(* LS Electric XG5000 project: Stride_IOLink_EIP_FB *)
(* project contains a function block for communicating with Automationdirect's IO-Link masters *)
(* PLC LSPLC *)
(* module base 0 slot 0: Input/Output Module:XEM-DN/DP32HP (DC 24V Input, Transistor Output, 32 Contacts) *)
(* module base 0 slot 1: Internal Positioning:XBF-PO06E (Open Collector Type, 6 Axis) *)
(* module base 0 slot 2: EtherNet/IP:XBL-EIPT (EtherNet/IP communication module, electrical) *)
VAR_GLOBAL
    Stride_IOLink_Input00 : ARRAY[0..393] OF BYTE; (* Input data for IO-Link master *)
    Stride_IOLink_Output00 : ARRAY[0..259] OF BYTE; (* Output data for IO-Link master *)
END_VAR

TYPE Contrinex_RLH_RFID_UDT : (* data type for Contrinex RLH-xxxPA-NIS RFID reader/writer with IO-Link interface. *)
STRUCT
    Status_Ready : BOOL; (* Will toggle state when command executed and new data is available *)
    Status_Error : BOOL; (* Command executed with error. *)
    Status_Tag_Present : BOOL; (* Tag present in range of transponder *)
    Status_Antenna_On : BOOL; (* Transponder antenna is powered *)
    Status_RSSI_Level : USINT; (* Signal level between transponder and tag. *)
    Status_Error_Code : USINT; (* ISO 15693 error code. 1: CommandNotSupported. 2: FormatError. 3: OptionNotSupported. 5: CommandProblem. 6: CommTagError. 15:TagError. 16: NoMemoryBlock. 18: BlockProtected. 27:AppLOGError. 30: TAGCommError. 255: AppGeneralError. *)
    Status_Alarm_1 : BOOL; (* Alarm1 active *)
    Status_Alarm_2 : BOOL; (* Alarm 2 active *)
    Status_Address : USINT; (* First transponder memory block address where the R/W command was executed *)
    Status_Command_Feedback : USINT; (* Feedback of command sent to transponder *)
    Status_Tag_UID : ARRAY[0..7] OF BYTE; (* Transponder unique ID number *)
    Status_Tag_In_Range_Time : DINT; (* Transponder in-range time in milliseconds *)
    Status_Tag_In_Range_Start_Time : DINT; (* Transponder in-range system start time in milliseconds *)
    Status_Ready_Last_Scan : BOOL; (* Last Scan Data for determining change of ready bit. *)
    Status_Read_Tag_Value : ARRAY[0..30] OF BYTE; (* data read from userspace on tag *)
    Control_Set_Tag_Value : ARRAY[0..30] OF BYTE; (* data to write to userspace on tag *)
    Received_Tag_ASCII : STRING; (* received transponder data, converted to ASCII for readability *)
    Set_Tag_ASCII : STRING; (* Optional ASCII string to send to transponder if readable text is desired. *)
    Control_Start_Operation : BOOL; (* Toggle to begin desired RFID operation (not used for Auto-Read or Auto-Write) *)
    Control_Switch_Off_Antenna : BOOL; (* Disables antenna when high *)
    Control_Command : USINT; (* command to send to transponder *)
    Control_NB_Block : USINT; (* number of transponder memory block to R/W *)
    Control_Address : USINT; (* first transponder memory block address where the R/W command will be executed. *)
    Control_Mode_Set_None : BOOL; (* Set to High to disable RFID functions *)
    Control_Mode_Set_Auto_Read : BOOL; (* Set to high to enable auto-read function. *)
    Control_Mode_Set_Auto_Write : BOOL; (* Set to high to enable auto-write function *)
    Control_Mode_Set_Read : BOOL; (* Set to high to attempt one single read *)
    Control_Mode_Set_Write : BOOL; (* Set to high to attempt one single write *)
    Control_Mode_Set_Read_Sys : BOOL; (* Set to high to enable tag UID and timings function *)
    Scans_Since_Tag_Last_Seen : UINT; (* Counter value to watch for absence of tag. *)
END_STRUCT;
END_TYPE

TYPE Murr_DIO_Hub_UDT : (* user data type for the Murrelektronik MVP12/MVP8 Digital Input/Output IO-Link hub *)
STRUCT
    Digital_Input : ARRAY[0..15] OF BOOL; (* Mapped Digital Inputs *)
    Digital_Output : ARRAY[0..15] OF BOOL; (* Mapped Digital Outputs *)
    Fault_Present : BOOL; (* Active if there is a fault with MURR dio hub *)
    Fault_IO_Point : INT; (* ID of channel experiencing a fault *)
END_STRUCT;
END_TYPE

TYPE Stride_IOLink_Port_UDT :
STRUCT
    Vendor_ID : UINT; (* IO-Link Vendor ID *)
    Device_ID : DINT; (* IO-Link Device ID *)
    Port_Status_Operate : BOOL; (* 1 = device is connected and active *)
    Port_Status_Error : BOOL; (* 1 = error or warning has occurred on this port *)
    Port_Status_Valid : BOOL; (* 1 = process data is valid *)
    Discrete_Input : ARRAY[0..1] OF BOOL; (* Physical Input pins *)
    Discrete_Output : ARRAY[0..1] OF BOOL; (* Physical Output pins *)
    Cyclic_Data_In : ARRAY[0..31] OF BYTE; (* process data from IO-Link device. *)
    Cyclic_Data_Out : ARRAY[0..31] OF BYTE; (* Control data to IO-Link device. *)
END_STRUCT;
END_TYPE

FUNCTION_BLOCK Contrinex_RFID_FB
(* Function block for Contrinex RLH-xxxPA-NIS RFID system *)
VAR_INPUT
    Enable : BOOL; (* Enable for function block *)
    Copy_SetTagASCII_to_ControlSetValue : BOOL; (* this will enable copying UserRFID.Set_Tag_ASCII to UserRFID.Control.Set_Tag_Value. *)
END_VAR
VAR_IN_OUT
    User_RFID : Contrinex_RLH_RFID_UDT; (* Data type for the Contrinex RFID module *)
    Port : Stride_IOLink_Port_UDT; (* variable for IO-Link master port. *)
END_VAR
VAR_OUTPUT
    Active : BOOL; (* Function block is active. *)
END_VAR
VAR
    InTemp : ARRAY[0..31] OF BYTE; (* temporary input array *)
    OutTemp : ARRAY[0..31] OF BYTE; (* temporary output array *)
    tempBool : BOOL; (* temporary bool storage *)
    tempDWord1 : DWORD; (* temporary dword storage *)
    tempWord1 : WORD; (* temporary word storage *)
    tempWord2 : WORD; (* temporary word storage *)
END_VAR
(*
AutomationDirect.com has provided this code for convenience. This sample code is provided "as-is" with no expressed or implied warranty and has not been thoroughly tested for all conditions and environments.  
While AutomationDirect.com makes every effort to provide error-free code that can be used as-is, it is the user's responsibility to completely test this code in operation to ensure it meets all system and safety requirements for the intended application or system.
 By loading and running this code, you are acknowledging the responsibility to completely test the code in your system before deployment.
*)
(***************************************************************************************************
	The 'Contrinex_RFID_FB' function block use one of the Port_X0 thru Port_X7 from Stride_IOLink_Master_FB.
		This function block separates the source data buffers for a Contrinex RLH RFID module that is connected to the given Port_XX that is passed in.
						
	***************************************************************************************************)
	
	IF (Enable = TRUE) THEN
		Active := TRUE;
		
		(* Map Status variables *)
		InTemp := ARY_MOVE(MOVE_NUM:=31, IN:=Port.Cyclic_Data_In, IN_INDX:=0, OUT_INDX:=0);
		
		User_RFID.Status_Command_Feedback.0  := InTemp[0].0;
		User_RFID.Status_Command_Feedback.1  := InTemp[0].1;
		User_RFID.Status_Command_Feedback.2  := InTemp[0].2;
		User_RFID.Status_Antenna_On  := InTemp[0].4;
		User_RFID.Status_Tag_Present  := InTemp[0].5;
		User_RFID.Status_Error  := InTemp[0].6;
		User_RFID.Status_Ready  := InTemp[0].7;
		
		User_RFID.Status_Alarm_1  := InTemp[1].0;
		User_RFID.Status_Alarm_2  := InTemp[1].1;
		User_RFID.Status_Error_Code.0  := InTemp[1].2;
		User_RFID.Status_Error_Code.1  := InTemp[1].3;
		User_RFID.Status_Error_Code.2  := InTemp[1].4;
		User_RFID.Status_Error_Code.3  := InTemp[1].5;
		User_RFID.Status_Error_Code.4  := InTemp[1].6;
		User_RFID.Status_Error_Code.5  := InTemp[1].7;
		
		User_RFID.Status_RSSI_Level :=  BYTE_TO_USINT(InTemp[2]);
		User_RFID.Status_Address := BYTE_TO_USINT(InTemp[3]);
		
		
		//control mode commands.
		IF (User_RFID.Control_Mode_Set_None = TRUE) THEN
			User_RFID.Control_Command := 0;
			User_RFID.Control_Mode_Set_None := FALSE;
		
		ELSIF (User_RFID.Control_Mode_Set_Auto_Read = TRUE) THEN
			User_RFID.Control_Command := 1;
			User_RFID.Control_Mode_Set_Auto_Read := FALSE;
		
		ELSIF (User_RFID.Control_Mode_Set_Auto_Write = TRUE) THEN
			User_RFID.Control_Command := 2;	
			User_RFID.Control_Mode_Set_Auto_Write := FALSE;
			
		ELSIF (User_RFID.Control_Mode_Set_Read = TRUE) THEN
			User_RFID.Control_Command := 3;		
			User_RFID.Control_Mode_Set_Read := FALSE;
		
		ELSIF ( User_RFID.Control_Mode_Set_Write = TRUE) THEN
			User_RFID.Control_Command := 4;		
		  	User_RFID.Control_Mode_Set_Write :=  FALSE;
		  	
		  ELSIF(User_RFID.Control_Mode_Set_Read_Sys = TRUE) THEN
		  	User_RFID.Control_Command := 5;	
		    User_RFID.Control_Mode_Set_Read_Sys := FALSE;
		    
		   END_IF; 
		
		//update last read tag when new data available.
		IF (User_RFID.Status_Command_Feedback = 1 OR User_RFID.Status_Command_Feedback = 3) AND ( (User_RFID.Status_Ready = TRUE AND User_RFID.Status_Ready_Last_Scan = FALSE) OR (User_RFID.Status_Ready_Last_Scan = TRUE AND User_RFID.Status_Ready = FALSE) ) THEN
			User_RFID.Status_Read_Tag_Value := ARY_MOVE(MOVE_NUM:=28, IN:=InTemp, IN_INDX:=4, OUT_INDX:=0);
		END_IF;
		
		//Convert received tag data to ASCII
		User_RFID.Received_Tag_ASCII :=BYTE_STRING(IN:=User_RFID.Status_Read_Tag_Value);
		
		
		//calculate 'tag-in-range' times and read tag UID
		IF (User_RFID.Status_Command_Feedback = 5) THEN
			
			tempWord1 := BYTE_WORD(LOW:=InTemp[27], HIGH:=InTemp[26]);
			tempWord2 :=BYTE_WORD(LOW:=InTemp[25], HIGH:=InTemp[24]);
			tempDWord1 := WORD_DWORD(LOW:=tempWord1, HIGH:= tempWord2);
			User_RFID.Status_Tag_In_Range_Time := DWORD_TO_DINT(IN:= tempDWord1);
			
			tempWord1 := BYTE_WORD(LOW:=InTemp[19], HIGH:=InTemp[18]);
			tempWord2 :=BYTE_WORD(LOW:=InTemp[17], HIGH:=InTemp[16]);
			tempDWord1 := WORD_DWORD(LOW:=tempWord1, HIGH:= tempWord2);
			User_RFID.Status_Tag_In_Range_Start_Time := DWORD_TO_DINT(IN:= tempDWord1);
			
			User_RFID.Status_Tag_UID := ARY_MOVE(MOVE_NUM:=8, IN:=InTemp, IN_INDX:=5, OUT_INDX:=0);
			
		END_IF;
		
		
		//Clear read tag data when tag isn't present for 50 scans
		IF (User_RFID.Status_Tag_Present = TRUE) THEN
			User_RFID.Scans_Since_Tag_Last_Seen := 0;
		ELSE
			User_RFID.Scans_Since_Tag_Last_Seen := User_RFID.Scans_Since_Tag_Last_Seen + 1;
		END_IF;
		
		IF (User_RFID.Scans_Since_Tag_Last_Seen > 50) THEN
			tempBool := ARY_FLL(DATA:=0, SRC:=User_RFID.Status_Read_Tag_Value, INDX:=0, LEN:=28);
			tempBool := ARY_FLL(DATA:=0, SRC:=User_RFID.Status_Tag_UID, INDX:=0, LEN:=8);
		END_IF;
		
		
		//when write command active, copy desired tag value to output data
		IF (User_RFID.Status_Command_Feedback =  4) OR (User_RFID.Status_Command_Feedback = 2) THEN
			OutTemp := ARY_MOVE(MOVE_NUM:=28, IN:=User_RFID.Control_Set_Tag_Value, IN_INDX:=0, OUT_INDX:=4); 
		END_IF;
		
		//copy string into set array if enabled
		IF (Copy_SetTagASCII_to_ControlSetValue = TRUE) THEN
			User_RFID.Control_Set_Tag_Value :=STRING_BYTE(IN:=User_RFID.Set_Tag_ASCII);
		END_IF;	
		
		//Pack commands into first command byte.
		OutTemp[0].0  := User_RFID.Control_Command.0;
		OutTemp[0].1  := User_RFID.Control_Command.1;
		OutTemp[0].2  := User_RFID.Control_Command.2;
		OutTemp[0].4  := User_RFID.Control_Switch_Off_Antenna;
		OutTemp[0].7  := User_RFID.Control_Start_Operation;
		
		
		//pack memory block target size into second command byte.
		OutTemp[1].0  := User_RFID.Control_NB_Block.0;
		OutTemp[1].1  := User_RFID.Control_NB_Block.1;
		OutTemp[1].2  := User_RFID.Control_NB_Block.2;
		
		//copy target memory address start point into fourth command byte
		OutTemp[3]  := USINT_TO_BYTE(User_RFID.Control_Address);
		
		//copy tag ready bit value to last-scan value
		User_RFID.Status_Ready_Last_Scan :=  User_RFID.Status_Ready;
		
		//map outputs to port
		Port.Cyclic_Data_Out := ARY_MOVE(MOVE_NUM:=32, IN:=OutTemp, IN_INDX:=0, OUT_INDX:=0);
	
		
	ELSE
		Active := FALSE;
		
	END_IF;
END_FUNCTION_BLOCK

FUNCTION_BLOCK Murr_DIO_Hub_FB
(* function block for mapping data from Murrelektronik MVP12/MVP8 Digital Input/Output IO-Link hub *)
VAR_INPUT
    Enable : BOOL; (* enable function block *)
END_VAR
VAR_IN_OUT
    DIO_Hub : Murr_DIO_Hub_UDT; (* variable for MURR DIO Hub *)
    Port : Stride_IOLink_Port_UDT; (* variable for IO-Link master port. *)
END_VAR
VAR_OUTPUT
    Active : BOOL; (* function block is active *)
END_VAR
VAR
    InTemp : ARRAY[0..31] OF BYTE; (* temporary input array *)
    OutTemp : ARRAY[0..31] OF BYTE; (* temporary output array *)
END_VAR
(*
AutomationDirect.com has provided this code for convenience. This sample code is provided "as-is" with no expressed or implied warranty and has not been thoroughly tested for all conditions and environments.  
While AutomationDirect.com makes every effort to provide error-free code that can be used as-is, it is the user's responsibility to completely test this code in operation to ensure it meets all system and safety requirements for the intended application or system.
 By loading and running this code, you are acknowledging the responsibility to completely test the code in your system before deployment.
*)
(***************************************************************************************************
	The 'Murr_DIO_Hub_FB' function block use one of the Port_X0 thru Port_X7 from Stride_IOLink_Master_FB.
		This function block separates the source data buffers for a Murr DIO Hub that is connected to the given Port_XX that is passed in.
						
	***************************************************************************************************)
	
IF (Enable = TRUE) THEN		
	Active := TRUE;
	
	//map inputs
	InTemp := ARY_MOVE(MOVE_NUM:=31, IN:=Port.Cyclic_Data_In, IN_INDX:=0, OUT_INDX:=0);
	
	DIO_Hub.Digital_Input[0] := InTemp[0].0;
	DIO_Hub.Digital_Input[1] := InTemp[0].1;
	DIO_Hub.Digital_Input[2] := InTemp[0].2;
	DIO_Hub.Digital_Input[3] := InTemp[0].3;
	DIO_Hub.Digital_Input[4] := InTemp[0].4;
	DIO_Hub.Digital_Input[5] := InTemp[0].5;
	DIO_Hub.Digital_Input[6] := InTemp[0].6;
	DIO_Hub.Digital_Input[7] := InTemp[0].7;
	DIO_Hub.Digital_Input[8] := InTemp[1].0;
	DIO_Hub.Digital_Input[9] := InTemp[1].1;
	DIO_Hub.Digital_Input[10] := InTemp[1].2;
	DIO_Hub.Digital_Input[11] := InTemp[1].3;
	DIO_Hub.Digital_Input[12] := InTemp[1].4;
	DIO_Hub.Digital_Input[13] := InTemp[1].5;
	DIO_Hub.Digital_Input[14] := InTemp[1].6;
	DIO_Hub.Digital_Input[15] := InTemp[1].7;	
	
	DIO_Hub.Fault_Present := InTemp[2].0;
	
	// map io point number that has a fault
	DIO_Hub.Fault_IO_Point.0 := InTemp[2].3;
	DIO_Hub.Fault_IO_Point.1 := InTemp[2].4;
	DIO_Hub.Fault_IO_Point.2 := InTemp[2].5;
	DIO_Hub.Fault_IO_Point.3 := InTemp[2].6;
	
	//map outputs from DIO Hub to OutTemp
	OutTemp[0].0 := DIO_Hub.Digital_Output[0];
	OutTemp[0].1 := DIO_Hub.Digital_Output[1];
	OutTemp[0].2 := DIO_Hub.Digital_Output[2];
	OutTemp[0].3 := DIO_Hub.Digital_Output[3];
	OutTemp[0].4 := DIO_Hub.Digital_Output[4];
	OutTemp[0].5 := DIO_Hub.Digital_Output[5];
	OutTemp[0].6 := DIO_Hub.Digital_Output[6];
	OutTemp[0].7 := DIO_Hub.Digital_Output[7];
	OutTemp[1].0 := DIO_Hub.Digital_Output[8];
	OutTemp[1].1 := DIO_Hub.Digital_Output[9];
	OutTemp[1].2 := DIO_Hub.Digital_Output[10];
	OutTemp[1].3 := DIO_Hub.Digital_Output[11];
	OutTemp[1].4 := DIO_Hub.Digital_Output[12];
	OutTemp[1].5 := DIO_Hub.Digital_Output[13];
	OutTemp[1].6 := DIO_Hub.Digital_Output[14];
	OutTemp[1].7 := DIO_Hub.Digital_Output[15];
	
	
	
	
	//map outputs to port
	Port.Cyclic_Data_Out := ARY_MOVE(MOVE_NUM:=32, IN:=OutTemp, IN_INDX:=0, OUT_INDX:=0);
	
	
ELSE
	Active := FALSE;
	
END_IF;
END_FUNCTION_BLOCK

FUNCTION_BLOCK Stride_IOLink_Master_FB
(* function block for mapping data from Stride Ethernet/IP IO-Link master *)
VAR_INPUT
    Enable : BOOL; (* Enable the function block *)
    Source_InputData : ARRAY[0..393] OF BYTE; (* Input data from the EtherNet/IP IO-Link master *)
END_VAR
VAR_IN_OUT
    Source_OutputData : ARRAY[0..259] OF BYTE; (* Output data from the EtherNet/IP IO-Link master *)
    Port_X0 : Stride_IOLink_Port_UDT; (* Port X0 of IO-Link master *)
    Port_X1 : Stride_IOLink_Port_UDT; (* Port X1 of IO-Link master *)
    Port_X2 : Stride_IOLink_Port_UDT; (* Port X2 of IO-Link master *)
    Port_X3 : Stride_IOLink_Port_UDT; (* Port X3 of IO-Link master *)
    Port_X4 : Stride_IOLink_Port_UDT; (* Port X4 of IO-Link master *)
    Port_X5 : Stride_IOLink_Port_UDT; (* Port X5 of IO-Link master *)
    Port_X6 : Stride_IOLink_Port_UDT; (* Port X6 of IO-Link master *)
    Port_X7 : Stride_IOLink_Port_UDT; (* Port X7 of IO-Link master *)
END_VAR
VAR_OUTPUT
    Active : BOOL; (* status that function block is active *)
END_VAR
VAR
    InputStatus : ARRAY[0..7] OF BYTE; (* input status data *)
    InTemp : ARRAY[0..393] OF BYTE; (* temporary input buffer to copy Source_InputData too. *)
    OutTemp : ARRAY[0..259] OF BYTE; (* temporary output buffer to copy to Source_OutputData *)
    WTemp1 : WORD; (* temporary word 1 *)
    WTemp2 : WORD; (* temporary word 2 *)
END_VAR
(*
AutomationDirect.com has provided this code for convenience. This sample code is provided "as-is" with no expressed or implied warranty and has not been thoroughly tested for all conditions and environments.  
While AutomationDirect.com makes every effort to provide error-free code that can be used as-is, it is the user's responsibility to completely test this code in operation to ensure it meets all system and safety requirements for the intended application or system.
 By loading and running this code, you are acknowledging the responsibility to completely test the code in your system before deployment.
*)
(***************************************************************************************************
	The 'Stride_IOLink_Master_FB' function block uses data type BYTE for Source_InputData and Source_OutputData.
		This function block separates the source data buffers into the individual ports of X0 thru X7.
		
									Data type:: BYTE
									Input Size: 394 bytes
									Output Size: 260 bytes
									EDS File: SIOL_EI8B_EIP_Rev_1_1.eds
									
	***************************************************************************************************)
	
IF (Enable = TRUE) THEN		
	Active := TRUE;	
	
	//copy Source_InputData to temporary local one
	InTemp := ARY_MOVE(MOVE_NUM:=394, IN:=Source_InputData, IN_INDX:=0, OUT_INDX:=0);
	

	//Port X0 mapping
	Port_X0.Discrete_Input[0] := InTemp[0].0;
	Port_X0.Discrete_Input[1] := InTemp[0].1;
	OutTemp[0].0 := Port_X0.Discrete_Output[0];
	OutTemp[0].1 :=Port_X0.Discrete_Output[1];
	
	Port_X0.Cyclic_Data_In := ARY_MOVE(MOVE_NUM:=32, IN:=InTemp, IN_INDX:=10, OUT_INDX:=0);
	InputStatus := ARY_MOVE(MOVE_NUM:=8, IN:=InTemp, IN_INDX:=42, OUT_INDX:=0);
	OutTemp := ARY_MOVE(MOVE_NUM:=32, IN:=Port_X0.Cyclic_Data_Out, IN_INDX:=0, OUT_INDX:=2);
	
	Port_X0.Port_Status_Operate := InputStatus[0].5;
	Port_X0.Port_Status_Error :=  InputStatus[0].6;
	Port_X0.Port_Status_Valid := InputStatus[0].7;
	
	Port_X0.Vendor_ID := WORD_TO_UINT(BYTE_WORD(LOW:=InputStatus[2], HIGH:=InputStatus[3]));
	
	WTemp1 := BYTE_WORD(LOW:=InputStatus[4], HIGH:=InputStatus[5]);
	WTemp2 := BYTE_WORD(LOW:=InputStatus[6], HIGH:=InputStatus[7]);
	Port_X0.Device_ID := DWORD_TO_DINT(WORD_DWORD(LOW:=WTemp1, HIGH:=WTemp2));
	
	
	
	//Port X1 mapping
	Port_X1.Discrete_Input[0] := InTemp[0].2;
	Port_X1.Discrete_Input[1] := InTemp[0].3;
	OutTemp[0].2 := Port_X1.Discrete_Output[0];
	OutTemp[0].3 :=Port_X1.Discrete_Output[1];
	
	Port_X1.Cyclic_Data_In := ARY_MOVE(MOVE_NUM:=32, IN:=InTemp, IN_INDX:=50, OUT_INDX:=0);
	InputStatus := ARY_MOVE(MOVE_NUM:=8, IN:=InTemp, IN_INDX:=82, OUT_INDX:=0);
	OutTemp := ARY_MOVE(MOVE_NUM:=32, IN:=Port_X1.Cyclic_Data_Out, IN_INDX:=0, OUT_INDX:=34);
	
	Port_X1.Port_Status_Operate := InputStatus[0].5;
	Port_X1.Port_Status_Error :=  InputStatus[0].6;
	Port_X1.Port_Status_Valid := InputStatus[0].7;
	
	Port_X1.Vendor_ID := WORD_TO_UINT(BYTE_WORD(LOW:=InputStatus[2], HIGH:=InputStatus[3]));
	
	WTemp1 := BYTE_WORD(LOW:=InputStatus[4], HIGH:=InputStatus[5]);
	WTemp2 := BYTE_WORD(LOW:=InputStatus[6], HIGH:=InputStatus[7]);
	Port_X1.Device_ID := DWORD_TO_DINT(WORD_DWORD(LOW:=WTemp1, HIGH:=WTemp2));	
	
	
	
	//Port X2 mapping
	Port_X2.Discrete_Input[0] := InTemp[0].4;
	Port_X2.Discrete_Input[1] := InTemp[0].5;
	OutTemp[0].4 := Port_X2.Discrete_Output[0];
	OutTemp[0].5 :=Port_X2.Discrete_Output[1];
	
	Port_X2.Cyclic_Data_In := ARY_MOVE(MOVE_NUM:=32, IN:=InTemp, IN_INDX:=90, OUT_INDX:=0);
	InputStatus := ARY_MOVE(MOVE_NUM:=8, IN:=InTemp, IN_INDX:=122, OUT_INDX:=0);
	OutTemp := ARY_MOVE(MOVE_NUM:=32, IN:=Port_X2.Cyclic_Data_Out, IN_INDX:=0, OUT_INDX:=66);
	
	Port_X2.Port_Status_Operate := InputStatus[0].5;
	Port_X2.Port_Status_Error :=  InputStatus[0].6;
	Port_X2.Port_Status_Valid := InputStatus[0].7;
	
	Port_X2.Vendor_ID := WORD_TO_UINT(BYTE_WORD(LOW:=InputStatus[2], HIGH:=InputStatus[3]));
	
	WTemp1 := BYTE_WORD(LOW:=InputStatus[4], HIGH:=InputStatus[5]);
	WTemp2 := BYTE_WORD(LOW:=InputStatus[6], HIGH:=InputStatus[7]);
	Port_X2.Device_ID := DWORD_TO_DINT(WORD_DWORD(LOW:=WTemp1, HIGH:=WTemp2));	
	
	
	
	//Port X3 mapping
	Port_X3.Discrete_Input[0] := InTemp[0].6;
	Port_X3.Discrete_Input[1] := InTemp[0].7;
	OutTemp[0].6 := Port_X3.Discrete_Output[0];
	OutTemp[0].7 :=Port_X3.Discrete_Output[1];
	
	Port_X3.Cyclic_Data_In := ARY_MOVE(MOVE_NUM:=32, IN:=InTemp, IN_INDX:=130, OUT_INDX:=0);
	InputStatus := ARY_MOVE(MOVE_NUM:=8, IN:=InTemp, IN_INDX:=162, OUT_INDX:=0);
	OutTemp := ARY_MOVE(MOVE_NUM:=32, IN:=Port_X3.Cyclic_Data_Out, IN_INDX:=0, OUT_INDX:=98);
	
	Port_X3.Port_Status_Operate := InputStatus[0].5;
	Port_X3.Port_Status_Error :=  InputStatus[0].6;
	Port_X3.Port_Status_Valid := InputStatus[0].7;
	
	Port_X3.Vendor_ID := WORD_TO_UINT(BYTE_WORD(LOW:=InputStatus[2], HIGH:=InputStatus[3]));
	
	WTemp1 := BYTE_WORD(LOW:=InputStatus[4], HIGH:=InputStatus[5]);
	WTemp2 := BYTE_WORD(LOW:=InputStatus[6], HIGH:=InputStatus[7]);
	Port_X3.Device_ID := DWORD_TO_DINT(WORD_DWORD(LOW:=WTemp1, HIGH:=WTemp2));	
	
	
	
	//Port X4 mapping
	Port_X4.Discrete_Input[0] := InTemp[1].0;
	Port_X4.Discrete_Input[1] := InTemp[1].1;
	OutTemp[1].0 := Port_X4.Discrete_Output[0];
	OutTemp[1].1 :=Port_X4.Discrete_Output[1];
	
	Port_X4.Cyclic_Data_In := ARY_MOVE(MOVE_NUM:=32, IN:=InTemp, IN_INDX:=170, OUT_INDX:=0);
	InputStatus := ARY_MOVE(MOVE_NUM:=8, IN:=InTemp, IN_INDX:=202, OUT_INDX:=0);
	OutTemp := ARY_MOVE(MOVE_NUM:=32, IN:=Port_X4.Cyclic_Data_Out, IN_INDX:=0, OUT_INDX:=130);
	
	Port_X4.Port_Status_Operate := InputStatus[0].5;
	Port_X4.Port_Status_Error :=  InputStatus[0].6;
	Port_X4.Port_Status_Valid := InputStatus[0].7;
	
	Port_X4.Vendor_ID := WORD_TO_UINT(BYTE_WORD(LOW:=InputStatus[2], HIGH:=InputStatus[3]));
	
	WTemp1 := BYTE_WORD(LOW:=InputStatus[4], HIGH:=InputStatus[5]);
	WTemp2 := BYTE_WORD(LOW:=InputStatus[6], HIGH:=InputStatus[7]);
	Port_X4.Device_ID := DWORD_TO_DINT(WORD_DWORD(LOW:=WTemp1, HIGH:=WTemp2));		
	
	
	
	//Port X5 mapping
	Port_X5.Discrete_Input[0] := InTemp[1].2;
	Port_X5.Discrete_Input[1] := InTemp[1].3;
	OutTemp[1].2 := Port_X5.Discrete_Output[0];
	OutTemp[1].3 :=Port_X5.Discrete_Output[1];
	
	Port_X5.Cyclic_Data_In := ARY_MOVE(MOVE_NUM:=32, IN:=InTemp, IN_INDX:=210, OUT_INDX:=0);
	InputStatus := ARY_MOVE(MOVE_NUM:=8, IN:=InTemp, IN_INDX:=242, OUT_INDX:=0);
	OutTemp := ARY_MOVE(MOVE_NUM:=32, IN:=Port_X5.Cyclic_Data_Out, IN_INDX:=0, OUT_INDX:=162);
	
	Port_X5.Port_Status_Operate := InputStatus[0].5;
	Port_X5.Port_Status_Error :=  InputStatus[0].6;
	Port_X5.Port_Status_Valid := InputStatus[0].7;
	
	Port_X5.Vendor_ID := WORD_TO_UINT(BYTE_WORD(LOW:=InputStatus[2], HIGH:=InputStatus[3]));
	
	WTemp1 := BYTE_WORD(LOW:=InputStatus[4], HIGH:=InputStatus[5]);
	WTemp2 := BYTE_WORD(LOW:=InputStatus[6], HIGH:=InputStatus[7]);
	Port_X5.Device_ID := DWORD_TO_DINT(WORD_DWORD(LOW:=WTemp1, HIGH:=WTemp2));	
	

	//Port X6 mapping
	Port_X6.Discrete_Input[0] := InTemp[1].4;
	Port_X6.Discrete_Input[1] := InTemp[1].5;
	OutTemp[1].4 := Port_X6.Discrete_Output[0];
	OutTemp[1].5 :=Port_X6.Discrete_Output[1];
	
	Port_X6.Cyclic_Data_In := ARY_MOVE(MOVE_NUM:=32, IN:=InTemp, IN_INDX:=250, OUT_INDX:=0);
	InputStatus := ARY_MOVE(MOVE_NUM:=8, IN:=InTemp, IN_INDX:=282, OUT_INDX:=0);
	OutTemp := ARY_MOVE(MOVE_NUM:=32, IN:=Port_X6.Cyclic_Data_Out, IN_INDX:=0, OUT_INDX:=194);
	
	Port_X6.Port_Status_Operate := InputStatus[0].5;
	Port_X6.Port_Status_Error :=  InputStatus[0].6;
	Port_X6.Port_Status_Valid := InputStatus[0].7;
	
	Port_X6.Vendor_ID := WORD_TO_UINT(BYTE_WORD(LOW:=InputStatus[2], HIGH:=InputStatus[3]));
	
	WTemp1 := BYTE_WORD(LOW:=InputStatus[4], HIGH:=InputStatus[5]);
	WTemp2 := BYTE_WORD(LOW:=InputStatus[6], HIGH:=InputStatus[7]);
	Port_X6.Device_ID := DWORD_TO_DINT(WORD_DWORD(LOW:=WTemp1, HIGH:=WTemp2));	
	
	
	//Port X7 mapping
	Port_X7.Discrete_Input[0] := InTemp[1].6;
	Port_X7.Discrete_Input[1] := InTemp[1].7;
	OutTemp[1].6 := Port_X7.Discrete_Output[0];
	OutTemp[1].7 :=Port_X7.Discrete_Output[1];
	
	Port_X7.Cyclic_Data_In := ARY_MOVE(MOVE_NUM:=32, IN:=InTemp, IN_INDX:=290, OUT_INDX:=0);
	InputStatus := ARY_MOVE(MOVE_NUM:=8, IN:=InTemp, IN_INDX:=322, OUT_INDX:=0);
	OutTemp := ARY_MOVE(MOVE_NUM:=32, IN:=Port_X7.Cyclic_Data_Out, IN_INDX:=0, OUT_INDX:=226);
	
	Port_X7.Port_Status_Operate := InputStatus[0].5;
	Port_X7.Port_Status_Error :=  InputStatus[0].6;
	Port_X7.Port_Status_Valid := InputStatus[0].7;
	
	Port_X7.Vendor_ID := WORD_TO_UINT(BYTE_WORD(LOW:=InputStatus[2], HIGH:=InputStatus[3]));
	
	WTemp1 := BYTE_WORD(LOW:=InputStatus[4], HIGH:=InputStatus[5]);
	WTemp2 := BYTE_WORD(LOW:=InputStatus[6], HIGH:=InputStatus[7]);
	Port_X7.Device_ID := DWORD_TO_DINT(WORD_DWORD(LOW:=WTemp1, HIGH:=WTemp2));	

	
	
	//copy temporary output buffer to Source_OutputData
	Source_OutputData  := ARY_MOVE(MOVE_NUM:=260, IN:=OutTemp, IN_INDX:=0, OUT_INDX:=0); 
	
ELSE
	Active := FALSE;
	
END_IF;
END_FUNCTION_BLOCK

PROGRAM NewProgram (* task: Scan Program *)
VAR_EXTERNAL
    IOLink00_Port_X0 : Stride_IOLink_Port_UDT; (* Master00 port x0 *)
    IOLink00_Port_X1 : Stride_IOLink_Port_UDT; (* master00 port x1 *)
    IOLink00_Port_X2 : Stride_IOLink_Port_UDT; (* master00 port x2 *)
    IOLink00_Port_X3 : Stride_IOLink_Port_UDT; (* master00 port x3 *)
    IOLink00_Port_X4 : Stride_IOLink_Port_UDT; (* master00 port x4 *)
    IOLink00_Port_X5 : Stride_IOLink_Port_UDT; (* master00 port x5 *)
    IOLink00_Port_X6 : Stride_IOLink_Port_UDT; (* master00 port x6 *)
    IOLink00_Port_X7 : Stride_IOLink_Port_UDT; (* master00 port x7 *)
    Stride_IOLink_Input00 : ARRAY[0..393] OF BYTE; (* Input data for IO-Link master *)
    Stride_IOLink_Output00 : ARRAY[0..259] OF BYTE; (* Output data for IO-Link master *)
END_VAR
VAR
    Master00_INST : Stride_IOLink_Master_FB; (* instance of IO-Link master fb *)
END_VAR

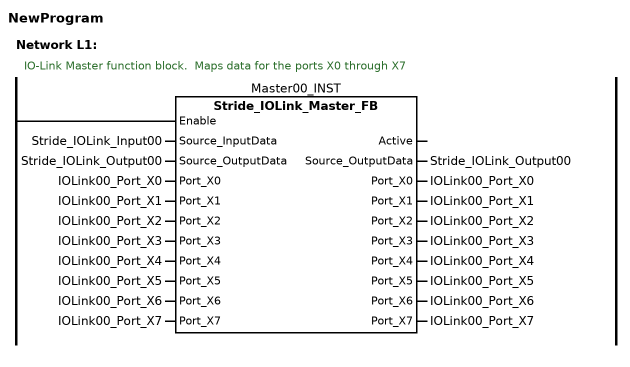
(* IO-Link Master function block.  Maps data for the ports X0 through X7 *)
(* Rung L1 *)
Master00_INST(Enable := TRUE, Source_InputData := Stride_IOLink_Input00, Source_OutputData := Stride_IOLink_Output00, Port_X0 := IOLink00_Port_X0, Port_X1 := IOLink00_Port_X1, Port_X2 := IOLink00_Port_X2, Port_X3 := IOLink00_Port_X3, Port_X4 := IOLink00_Port_X4, Port_X5 := IOLink00_Port_X5, Port_X6 := IOLink00_Port_X6, Port_X7 := IOLink00_Port_X7, Source_OutputData => Stride_IOLink_Output00, Port_X0 => IOLink00_Port_X0, Port_X1 => IOLink00_Port_X1, Port_X2 => IOLink00_Port_X2, Port_X3 => IOLink00_Port_X3, Port_X4 => IOLink00_Port_X4, Port_X5 => IOLink00_Port_X5, Port_X6 => IOLink00_Port_X6, Port_X7 => IOLink00_Port_X7);
END_PROGRAM